(* CODESYS project Lauda.library
   Company: Ziga Javornik
   DefaultNamespace: ZigaLibs.Lauda
   Version: 0.0.2.2
   Placeholder: ZigaLibs.Lauda
   Author: Ziga Javornik
   Description: Various Lauda device implementations.
   Title: ZigaLibs.Lauda

Project tree, tasks and I/O mapping:
  libraries: Tc2_Standard, * (Beckhoff Automation GmbH); Tc2_System, * (Beckhoff Automation GmbH); Tc2_TcpIp, * (Beckhoff Automation GmbH); Tc2_Utilities, * (Beckhoff Automation GmbH); Tc3_Module, * (Beckhoff Automation GmbH); TcUnit, 1.3.1 (www.tcunit.org); ZigaLibs.Core, 0.0.3.7 (Ziga Javornik); TcpIp, 0.0.2.2 (Ziga Javornik); ZigaLibs.Logging, * (Ziga Javornik)
  GVLs/
  SOURCE/
    Lauda Pro P20/
      DUTs/
        Commands/
          Read/
            Command groups/
              data type ST_LaudaReadCommands_ActuatingSignal
              data type ST_LaudaReadCommands_Control
              data type ST_LaudaReadCommands_ControlParameters
              data type ST_LaudaReadCommands_Cooling
              data type ST_LaudaReadCommands_FillLevel
              data type ST_LaudaReadCommands_Pump
              data type ST_LaudaReadCommands_Rights
              data type ST_LaudaReadCommands_Safety
              data type ST_LaudaReadCommands_Status
              data type ST_LaudaReadCommands_SwVersions
              data type ST_LaudaReadCommands_Temperature
            data type ST_LaudaReadCommands
          Write/
            Command groups/
              data type ST_LaudaWriteCommands_Control
              data type ST_LaudaWriteCommands_ControlParameters
              data type ST_LaudaWriteCommands_Cooling
              data type ST_LaudaWriteCommands_Pump
              data type ST_LaudaWriteCommands_Rights
              data type ST_LaudaWriteCommands_Safety
              data type ST_LaudaWriteCommands_Status
              data type ST_LaudaWriteCommands_Temperature
            data type ST_LaudaWriteCommands
          data type ST_LaudaCommands
        Errors/
          data type E_LaudaResponseError
          data type ST_LaudaFaults
          data type ST_LaudaReadWriteError
          data type ST_LaudaResponseErrors
        Parameters/
          data type ST_LaudaActualValuesCollection
          data type ST_LaudaCommParameters
        States/
          data type E_LaudaParameterReadState
          data type E_LaudaParameterWriteState
          data type E_ReadWriteStep
      POUs/
        Helpers/
          function block FB_LaudaCommandGenerator [ST]: KeyboardMasterLock, KeyboardMasterUnlock, KeyboardRemoteUnitLock, KeyboardRemoteUnitUnlock, SafetyActivate, SafetyDeactivate, SetPumpStage, SetTemperature, Start, Stop
          program LaudaHelper [ST]: AddSuffix, GenerateComand, ParseLaudaFaultDiagnosis, ParseResponseError, RemoveSuffix, ValidateReadCommandResponse, ValidateSendCommandResponse, Commands, ResponseErrors
        function block FB_LaudaPro_P20 [ST]: FB_init, AddToErrorBuffer, DequeueCommand, EnqueueCommand, ActualValues, CommParameters, DeviceFaultDiagnosis, Error, ErrorBuffer, Faults, TcpIpConnectionEstablished
  TESTS/
    Test suites/
      function block FB_LaudaHelperTests [ST]: Test01_AddSuffix, Test02_RemoveSuffix, Test03_ValidateReadCommandResponse, Test04_ValidateSendCommandResponse, Test05_ParseFault, Test06_ParseResponseError
    program PRG_TESTS [ST]
*)

// SOURCE/Lauda Pro P20/DUTs/Commands/Read/Command groups/ST_LaudaReadCommands_ActuatingSignal
TYPE ST_LaudaReadCommands_ActuatingSignal :
STRUCT
	Value	: STRING := 'IN_PV_06';
END_STRUCT
END_TYPE

// SOURCE/Lauda Pro P20/DUTs/Commands/Read/Command groups/ST_LaudaReadCommands_Control
TYPE ST_LaudaReadCommands_Control :
STRUCT
	SetpointOffset	: STRING := 'IN_PAR_14_';
	ControlVariable	: STRING := 'IN_MODE_01';
	OffsetSource	: STRING := 'IN_MODE_04';
END_STRUCT
END_TYPE

// SOURCE/Lauda Pro P20/DUTs/Commands/Read/Command groups/ST_LaudaReadCommands_ControlParameters
TYPE ST_LaudaReadCommands_ControlParameters :
STRUCT
END_STRUCT
END_TYPE

// SOURCE/Lauda Pro P20/DUTs/Commands/Read/Command groups/ST_LaudaReadCommands_Cooling
TYPE ST_LaudaReadCommands_Cooling :
STRUCT
	CoolingMode	: STRING := 'IN_SP_02';
END_STRUCT
END_TYPE

// SOURCE/Lauda Pro P20/DUTs/Commands/Read/Command groups/ST_LaudaReadCommands_FillLevel
TYPE ST_LaudaReadCommands_FillLevel :
STRUCT
	BathLevel	: STRING := 'IN_PV_05';
END_STRUCT
END_TYPE

// SOURCE/Lauda Pro P20/DUTs/Commands/Read/Command groups/ST_LaudaReadCommands_Pump
TYPE ST_LaudaReadCommands_Pump :
STRUCT
	FlowRate	: STRING := 'IN_PV_07';
	PowerStage	: STRING := 'IN_SP_01';
END_STRUCT
END_TYPE

// SOURCE/Lauda Pro P20/DUTs/Commands/Read/Command groups/ST_LaudaReadCommands_Rights
TYPE ST_LaudaReadCommands_Rights :
STRUCT
	KeyboardMaster_Locked				: STRING := 'IN_MODE_00_';
	KeyboardRemoveControlUnit_Locked	: STRING := 'IN_MODE_03';
END_STRUCT
END_TYPE

// SOURCE/Lauda Pro P20/DUTs/Commands/Read/Command groups/ST_LaudaReadCommands_Safety
TYPE ST_LaudaReadCommands_Safety :
STRUCT
	CommTimeoutViaInterface : STRING := 'IN_SP_08';
	SafetyModeActive		: STRING := 'IN_MODE_06';
END_STRUCT
END_TYPE

// SOURCE/Lauda Pro P20/DUTs/Commands/Read/Command groups/ST_LaudaReadCommands_Status
TYPE ST_LaudaReadCommands_Status :
STRUCT
	StandBy			: STRING := 'IN_MODE_02';
	DeviceType		: STRING := 'TYPE';
	DeviceStatus	: STRING := 'STATUS';
	FaultDiagnosis	: STRING := 'STAT';
END_STRUCT
END_TYPE

// SOURCE/Lauda Pro P20/DUTs/Commands/Read/Command groups/ST_LaudaReadCommands_SwVersions
TYPE ST_LaudaReadCommands_SwVersions :
STRUCT
	ControlSyste							: STRING := 'VERSION_R';
	ProtectionSystem						: STRING := 'VERSION_S';
	RemoteControl							: STRING := 'VERSION_B';
	CoolingSystem							: STRING := 'VERSION_T';
	AnalogInterfaceModule					: STRING := 'VERSION_A';
	RS232_422_Profibus_Profinet				: STRING := 'VERSION_V';
	EtherCAT								: STRING := 'VERSION_Z';
	ContactInterace							: STRING := 'VERSION_D';
	SolenoidValveForCoolingWater			: STRING := 'VERSION_M_0';
	SolenoidValveForAutomaticFillingDevice	: STRING := 'VERSION_M_1';
	SolenoidValveForConstantLevelDevice		: STRING := 'VERSION_M_2';
	SolenoidValve_ShutOffValve1				: STRING := 'VERSION_M_3';
	SolenoidValve_ShutOffValve2				: STRING := 'VERSION_M_4';
	ExternalPT100_interface1				: STRING := 'VERSION_E';
END_STRUCT
END_TYPE

// SOURCE/Lauda Pro P20/DUTs/Commands/Read/Command groups/ST_LaudaReadCommands_Temperature
TYPE ST_LaudaReadCommands_Temperature :
STRUCT
	TemperatureSetpoint				: STRING	 := 'IN_SP_00';
	BathTemperatureOutflow_01C		: STRING	 := 'IN_PV_00';
	BathTemperatureOutflow_001C		: STRING	 := 'IN_PV_10';
	QueryControlledTemperature		: STRING	 := 'IN_PV_01';
	ExternalTemperature_Pt_C		: STRING	 := 'IN_PV_03';
	ExternalTemperature_AnalogInput	: STRING	 := 'IN_PV_04';
	ExternalTemperature_Pt_001_C	: STRING	 := 'IN_PV_13';
	OvertemperatureTurnoffPoint_Tmax: STRING	 := 'IN_SP_03';
	OutflowLimmitHigh				: STRING	 := 'IN_SP_04';
	OutflowLimmitLow				: STRING	 := 'IN_SP_05';
	SafetyModeTemperature 			: STRING	 := 'IN_SP_07';
END_STRUCT
END_TYPE

// SOURCE/Lauda Pro P20/DUTs/Commands/Read/ST_LaudaReadCommands
TYPE ST_LaudaReadCommands :
STRUCT
	Temperature			: ST_LaudaReadCommands_Temperature;
	Pump				: ST_LaudaReadCommands_Pump;
	FillLevel			: ST_LaudaReadCommands_FillLevel;
	ActuatingSignal		: ST_LaudaReadCommands_ActuatingSignal;
	Cooling				: ST_LaudaReadCommands_Cooling;
	Safety				: ST_LaudaReadCommands_Safety;
	ControlParameters	: ST_LaudaReadCommands_ControlParameters;
	Control				: ST_LaudaReadCommands_Control;
	Rights				: ST_LaudaReadCommands_Rights;
	Status				: ST_LaudaReadCommands_Status;
	SwVersion			: ST_LaudaReadCommands_SwVersions;	
END_STRUCT
END_TYPE

// SOURCE/Lauda Pro P20/DUTs/Commands/Write/Command groups/ST_LaudaWriteCommands_Control
TYPE ST_LaudaWriteCommands_Control :
STRUCT
	SetpointOffset	: STRING := 'OUT_PAR_14_';
	ControlVariable	: STRING := 'OUT_MODE_01_X';
	OffsetSource	: string := 'OUT_MODE_04_X';
END_STRUCT
END_TYPE

// SOURCE/Lauda Pro P20/DUTs/Commands/Write/Command groups/ST_LaudaWriteCommands_ControlParameters
TYPE ST_LaudaWriteCommands_ControlParameters :
STRUCT
	Xp						: STRING := 'OUT_PAR_00_';
	Tn						: STRING := 'OUT_PAR_01_';
	Tv						: STRING := 'OUT_PAR_02_';
	Td						: STRING := 'OUT_PAR_03_';
	KpE						: STRING := 'OUT_PAR_04_';
	TnE						: STRING := 'OUT_PAR_05_';
	TvE						: STRING := 'OUT_PAR_06_';
	TdE						: STRING := 'OUT_PAR_07_';
	CorrectionLimitation	: STRING := 'OUT_PAR_09_';
	XpF						: STRING := 'OUT_PAR_10_';
	Prop_E					: STRING := 'OUT_PAR_15_';
END_STRUCT
END_TYPE

// SOURCE/Lauda Pro P20/DUTs/Commands/Write/Command groups/ST_LaudaWriteCommands_Cooling
TYPE ST_LaudaWriteCommands_Cooling :
STRUCT
	CoolingMode	: STRING := 'OUT_SP_02';
END_STRUCT
END_TYPE

// SOURCE/Lauda Pro P20/DUTs/Commands/Write/Command groups/ST_LaudaWriteCommands_Pump
TYPE ST_LaudaWriteCommands_Pump :
STRUCT
	Stage	: STRING := 'OUT_SP_01_';	// Pump stage 1-6 or 1-8 (device specific)
END_STRUCT
END_TYPE

// SOURCE/Lauda Pro P20/DUTs/Commands/Write/Command groups/ST_LaudaWriteCommands_Rights
TYPE ST_LaudaWriteCommands_Rights :
STRUCT
	KeyboardMaster_UnlockLock				: STRING := 'OUT_MODE_00_';
	KeyboardRemoteControlUnit_UnlockLock	: STRING := 'OUT_MODE_03_';
END_STRUCT
END_TYPE

// SOURCE/Lauda Pro P20/DUTs/Commands/Write/Command groups/ST_LaudaWriteCommands_Safety
TYPE ST_LaudaWriteCommands_Safety :
STRUCT
	CommTimeoutViaInterface : STRING := 'OUT_SP_08_';
	ActivateSafetyMode		: STRING := 'OUT_MODE_06_';
END_STRUCT
END_TYPE

// SOURCE/Lauda Pro P20/DUTs/Commands/Write/Command groups/ST_LaudaWriteCommands_Status
TYPE ST_LaudaWriteCommands_Status :
STRUCT
	Start	: STRING := 'START';
	Stop	: STRING := 'STOP';
END_STRUCT
END_TYPE

// SOURCE/Lauda Pro P20/DUTs/Commands/Write/Command groups/ST_LaudaWriteCommands_Temperature
TYPE ST_LaudaWriteCommands_Temperature :
STRUCT
	TemperatureSet				: STRING := 'OUT_SP_00_';
	ActualExternalTemperature	: STRING := 'OUT_PV_05_';
	OutflowLimmitHigh			: STRING := 'OUT_SP_04_';
	OutflowLimmitLow			: STRING := 'OUT_SP_05_';
	SafetyModeTemperature		: STRING := 'OUT_SP_07_';
END_STRUCT
END_TYPE

// SOURCE/Lauda Pro P20/DUTs/Commands/Write/ST_LaudaWriteCommands
TYPE ST_LaudaWriteCommands :
STRUCT
	Temperature			: ST_LaudaWriteCommands_Temperature;
	Control				: ST_LaudaWriteCommands_Control;
	ControlParameters	: ST_LaudaWriteCommands_ControlParameters;
	Cooling				: ST_LaudaWriteCommands_Cooling;
	Pump				: ST_LaudaWriteCommands_Pump;
	Rights				: ST_LaudaWriteCommands_Rights;
	Safety				: ST_LaudaWriteCommands_Safety;
	Status				: ST_LaudaWriteCommands_Status;
END_STRUCT
END_TYPE

// SOURCE/Lauda Pro P20/DUTs/Commands/ST_LaudaCommands
TYPE ST_LaudaCommands :
STRUCT
	Read	: ST_LaudaReadCommands;
	Write	: ST_LaudaWriteCommands;
END_STRUCT
END_TYPE

// SOURCE/Lauda Pro P20/DUTs/Errors/E_LaudaResponseError
{attribute 'qualified_only'}
{attribute 'strict'}
TYPE E_LaudaResponseError :
(
	NO_ERROR := 0,
	WRONG_ENTRY,
	WRONG_COMMAND,
	SYNTAX_ERROR,
	IMPERMISSABLE_VALUE,
	MODULE_OR_VALUE_NOT_AVAILABLE,
	ALL_SEGMENTS_IN_THE_PROGRAMMER_OCCUPIED,
	SETPOINT_NOT_POSSIBLE_WITH_ANALOG_SETPOINT_USED,
	EXTERNAL_TEMPERATURE_PROBE_MISSING,
	ANALOG_VALUE_NOT_PRESENT,
	SAFETY_MODE_CANT_START_IF_NOT_ENABLED,
	CANT_SET_VALUE_PROGRAMMER_RUNNING_OR_PAUSED,
	CANT_START_PROGRAMMER_ANALOG_SETPOINT_USED,
	CANT_ACTIVATE_FROM_SAFETY_MODE);
END_TYPE

// SOURCE/Lauda Pro P20/DUTs/Errors/ST_LaudaFaults
{attribute 'qualified_only'}
{attribute 'strict'}
TYPE ST_LaudaFaults :
STRUCT
	Error						: BOOL;
	Alarm						: BOOL;
	Warning						: BOOL;
	Overtemp					: BOOL;
	Sublevel					: BOOL;
	HigherLevel					: BOOL;
	ExternalControlValueMissing	: BOOL;
END_STRUCT
END_TYPE

// SOURCE/Lauda Pro P20/DUTs/Errors/ST_LaudaReadWriteError
{attribute 'qualified_only'}
{attribute 'strict'}
TYPE ST_LaudaReadWriteError :
STRUCT
	SendCommand			: STRING(100);
	ResponseErrorInfo	: E_LaudaResponseError;
END_STRUCT
END_TYPE

// SOURCE/Lauda Pro P20/DUTs/Errors/ST_LaudaResponseErrors
{attribute 'qualified_only'}
{attribute 'strict'}
{attribute 'to_string'}
TYPE ST_LaudaResponseErrors :
STRUCT
	WrongEntry	 								: STRING := 'ERR_2';
	WrongCommand								: STRING := 'ERR_3';
	SyntaxError	 								: STRING := 'ERR_5';
	ImpermissableValue	 						: STRING := 'ERR_6';
	ModuleOrValueNotAvailable					: STRING := 'ERR_8';
	AllSegmentsInTheProgrammerAreOccupied		: STRING := 'ERR_30';
	SetpointNotPossible_AnalogSetpointIsUsed	: STRING := 'ERR_31';
	ExternalTemperatureProbeMissing	 			: STRING := 'ERR_33';
	AnalogValueNotPresent	 					: STRING := 'ERR_34';
	SafetyModeCantBeStarted_ItIsNotEnabled	 	: STRING := 'ERR_35';
	CantSetValue_ProgrammerRunningOrPaused	 	: STRING := 'ERR_36';
	CantStartProgrammer_AnalogSetpointIsUsed	: STRING := 'ERR_37';
	CantActivateFromSafetyMode	 				: STRING := 'ERR_38';
END_STRUCT
END_TYPE

// SOURCE/Lauda Pro P20/DUTs/Parameters/ST_LaudaActualValuesCollection
{attribute 'qualified_only'}
{attribute 'strict'}
TYPE ST_LaudaActualValuesCollection :
STRUCT
	BathTemperature		: REAL;
	TemperatureSetpoint	: REAL;
	PumpStage			: UINT;
	StandBy				: BOOL;
	LiquidLevel			: UINT;
END_STRUCT
END_TYPE

// SOURCE/Lauda Pro P20/DUTs/Parameters/ST_LaudaCommParameters
{attribute 'qualified_only'}
{attribute 'strict'}
TYPE ST_LaudaCommParameters :
STRUCT
	ReadCycle		: TIME := T#500MS;			// Cyclic reading of certain values is executed within the interval defined by this parameter.
	ReconnectPeriod	: TIME := T#45S;			// Reconnect period for TCP/IP. Don't set too low (30s should be the lowest)
	Ipv4Address		: Tc2_System.T_IPv4Addr;	// IPV4 address of the device.
	Port			: UINT;						// Port of the device.
END_STRUCT
END_TYPE

// SOURCE/Lauda Pro P20/DUTs/States/E_LaudaParameterReadState
{attribute 'qualified_only'}
{attribute 'strict'}
TYPE E_LaudaParameterReadState :
(
	READY := 0,
	ACTUAL_TEMPERATURE_SETPOINT,
	BAH_OUTFLOW_TEMP,
	PUMP_STAGE,
	READ_ENABLE_STATE,
	OIL_LEVEL,
	FAULT_DIAGNOSIS,
	DONE
);
END_TYPE

// SOURCE/Lauda Pro P20/DUTs/States/E_LaudaParameterWriteState
{attribute 'qualified_only'}
{attribute 'strict'}
TYPE E_LaudaParameterWriteState :
(
	READY,
	SEND,
	AWAIT_RESPONSE,
	VALIDATE_RESPONSE,
	DONE
);
END_TYPE

// SOURCE/Lauda Pro P20/DUTs/States/E_ReadWriteStep
{attribute 'qualified_only'}
{attribute 'strict'}
TYPE E_ReadWriteStep :
(
	SEND,
	AWAIT_RESPONSE
);
END_TYPE

// SOURCE/Lauda Pro P20/POUs/Helpers/FB_LaudaCommandGenerator
FUNCTION_BLOCK FB_LaudaCommandGenerator
VAR_INPUT
END_VAR
VAR_OUTPUT
END_VAR
VAR
	_formatString	: Tc2_Utilities.FB_FormatString;
END_VAR

METHOD KeyboardMasterLock : T_MaxString
VAR_INPUT
END_VAR
KeyboardMasterLock := LaudaHelper.AddSuffix(CONCAT(
	STR1 := LaudaHelper.Commands.Write.Rights.KeyboardMaster_UnlockLock, 
	STR2 := '1'));
END_METHOD

METHOD KeyboardMasterUnlock : T_MaxString
VAR_INPUT
END_VAR
KeyboardMasterUnlock := LaudaHelper.AddSuffix(CONCAT(
	STR1 := LaudaHelper.Commands.Write.Rights.KeyboardMaster_UnlockLock, 
	STR2 := '0'));
END_METHOD

METHOD KeyboardRemoteUnitLock : Tc2_System.T_MaxString
VAR_INPUT
END_VAR
KeyboardRemoteUnitLock := LaudaHelper.AddSuffix(CONCAT(
	STR1 := LaudaHelper.Commands.Write.Rights.KeyboardRemoteControlUnit_UnlockLock, 
	STR2 := '1'));
END_METHOD

METHOD KeyboardRemoteUnitUnlock : Tc2_System.T_MaxString
VAR_INPUT
END_VAR
KeyboardRemoteUnitUnlock := LaudaHelper.AddSuffix(CONCAT(
	STR1 := LaudaHelper.Commands.Write.Rights.KeyboardRemoteControlUnit_UnlockLock, 
	STR2 := '0'));
END_METHOD

// Activates safety mode.
METHOD PUBLIC SafetyActivate : T_MaxString
VAR_INPUT
END_VAR
SafetyActivate := LaudaHelper.AddSuffix(
	sData := CONCAT(STR1 := LaudaHelper.Commands.Write.Safety.ActivateSafetyMode, STR2 := '1'));
END_METHOD

// Deactivates safety mode
METHOD PUBLIC SafetyDeactivate : T_MaxString
VAR_INPUT
END_VAR
SafetyDeactivate := LaudaHelper.AddSuffix(
	sData := CONCAT(STR1 := LaudaHelper.Commands.Write.Safety.ActivateSafetyMode, STR2 := '0'));
END_METHOD

// Sets pump stage, 1-6/9, depending on device specification
METHOD PUBLIC SetPumpStage : T_MaxString
VAR_INPUT
	nStage	: UINT;
END_VAR

VAR
	nPumpStageWithLimits	: UINT;
END_VAR
IF nStage < 1 THEN
	nPumpStageWithLimits := 1;
ELSIF nStage > 8 THEN
	nPumpStageWithLimits := 8;
ELSE
	nPumpStageWithLimits := nStage;
END_IF

SetPumpStage := LaudaHelper.AddSuffix(sData := Tc2_Standard.CONCAT(
		STR1 := LaudaHelper.Commands.Write.Pump.Stage, 
		STR2 := UINT_TO_STRING(nPumpStageWithLimits)));
END_METHOD

// Creates the command for temperature setting.
METHOD PUBLIC SetTemperature : T_maxstring
VAR_INPUT
	fTemperature	: REAL;	// Temperature setpoint to be set on the device.
END_VAR

VAR_INST
	errorID	: UDINT;
END_VAR
_formatString(
	sFormat := CONCAT(LaudaHelper.Commands.Write.Temperature.TemperatureSet, '%06.2f'),
	arg1 := Tc2_Utilities.F_REAL(in := fTemperature),
	nErrId => errorID);

SetTemperature := LaudaHelper.AddSuffix(_formatString.sOut);
END_METHOD

// Starts the device
METHOD PUBLIC Start : T_MaxString
Start := LaudaHelper.AddSuffix(sData := LaudaHelper.Commands.Write.Status.Start);
END_METHOD

// Stops the device
METHOD PUBLIC Stop : T_MaxString
Stop := LaudaHelper.AddSuffix(sData := LaudaHelper.Commands.Write.Status.Stop);
END_METHOD

END_FUNCTION_BLOCK

// SOURCE/Lauda Pro P20/POUs/Helpers/LaudaHelper
{attribute 'no_explicit_call' := 'Body contains no logic, calling methods only allowed.'}
{attribute 'hide_all_locals'}
// Provides various helper methods for easier communication with Lauda Pro device. 
// Program does not require being called, a simple access to methods is enough.
PROGRAM LaudaHelper
VAR
	_formatString			: FB_FormatString;
	_laudaCommandGenerator	: FB_LaudaCommandGenerator;	
	_commands				: ST_LaudaCommands;
	_responseErrors			: ST_LaudaResponseErrors;
END_VAR

VAR CONSTANT
	COMMAND_SUFFIX				: STRING := '$R$L';
	SEND_COMMAND_RESPONSE_OK	: STRING := 'OK';
	COMMAND_RESPONSE_ERROR		: STRING := 'ERR_'; 
END_VAR

// Adds suffix to the data command.
METHOD PUBLIC AddSuffix : Tc2_System.T_MaxString
VAR_INPUT
	sData	: Tc2_System.T_MaxString;
END_VAR
AddSuffix := Tc2_Standard.CONCAT(STR1 := sData, STR2 := COMMAND_SUFFIX);
END_METHOD

// Provides access to command generation methods.
METHOD PUBLIC GenerateComand : REFERENCE TO FB_LaudaCommandGenerator
VAR_INPUT
END_VAR
GenerateComand ref= _laudaCommandGenerator;
END_METHOD

// Parses the RAW data response for fault diagnosis and returns the faults structure.
METHOD ParseLaudaFaultDiagnosis : ST_LaudaFaults
VAR_INPUT
	sDiagnosisResposne	: Tc2_System.T_MaxString;
END_VAR
VAR
	sTmp		: Tc2_System.T_MaxString;
	nResponse	: BYTE;
	stFaults	: ST_LaudaFaults;
END_VAR

(*

*)
sTmp := RemoveSuffix(sData := sDiagnosisResposne);

stFaults.Error := INT_TO_BOOL(STRING_TO_INT(Tc2_Standard.MID(
	STR := sTmp,
	POS := 1, 
	LEN := 1)));

stFaults.Alarm := INT_TO_BOOL(STRING_TO_INT(Tc2_Standard.MID(
	STR := sTmp,
	POS := 2, 
	LEN := 1)));
	
stFaults.Warning := INT_TO_BOOL(STRING_TO_INT(Tc2_Standard.MID(
	STR := sTmp,
	POS := 3, 
	LEN := 1)));
	
stFaults.Overtemp := INT_TO_BOOL(STRING_TO_INT(Tc2_Standard.MID(
	STR := sTmp,
	POS := 4, 
	LEN := 1)));
	
stFaults.Sublevel := INT_TO_BOOL(STRING_TO_INT(Tc2_Standard.MID(
	STR := sTmp,
	POS := 5, 
	LEN := 1)));
	
stFaults.HigherLevel := INT_TO_BOOL(STRING_TO_INT(Tc2_Standard.MID(
	STR := sTmp,
	POS := 6, 
	LEN := 1)));
	
stFaults.ExternalControlValueMissing := INT_TO_BOOL(STRING_TO_INT(Tc2_Standard.MID(
	STR := sTmp,
	POS := 7, 
	LEN := 1)));
	
ParseLaudaFaultDiagnosis := stFaults;
END_METHOD

// Parses the error and returns the error message for further diagnosis
METHOD PUBLIC ParseResponseError : E_LaudaResponseError
VAR_INPUT
	Response	: Tc2_System.T_MaxString;
END_VAR
// Search the errors from highest to lowest to avoid case such as ERR_30 and you find it with ERR_3
// If success, return
IF Tc2_Standard.FIND(
	STR1 := Response, 
	STR2 := ResponseErrors.CantActivateFromSafetyMode) <> 0 
THEN
	ParseResponseError := E_LaudaResponseError.CANT_ACTIVATE_FROM_SAFETY_MODE;
	RETURN;
END_IF

IF Tc2_Standard.FIND(
	STR1 := Response, 
	STR2 := ResponseErrors.CantStartProgrammer_AnalogSetpointIsUsed) <> 0 
THEN
	ParseResponseError :=  E_LaudaResponseError.CANT_START_PROGRAMMER_ANALOG_SETPOINT_USED;
	RETURN;
END_IF

IF Tc2_Standard.FIND(
	STR1 := Response, 
	STR2 := ResponseErrors.CantSetValue_ProgrammerRunningOrPaused) <> 0 
THEN
	ParseResponseError :=  E_LaudaResponseError.CANT_SET_VALUE_PROGRAMMER_RUNNING_OR_PAUSED;
	RETURN;
END_IF

IF Tc2_Standard.FIND(
	STR1 := Response, 
	STR2 := ResponseErrors.SafetyModeCantBeStarted_ItIsNotEnabled) <> 0 
THEN
	ParseResponseError := E_LaudaResponseError.SAFETY_MODE_CANT_START_IF_NOT_ENABLED;
	RETURN;
END_IF

IF Tc2_Standard.FIND(
	STR1 := Response, 
	STR2 := ResponseErrors.AnalogValueNotPresent) <> 0 
THEN
	ParseResponseError := E_LaudaResponseError.ANALOG_VALUE_NOT_PRESENT;
	RETURN;
END_IF

IF Tc2_Standard.FIND(
	STR1 := Response, 
	STR2 := ResponseErrors.ExternalTemperatureProbeMissing) <> 0 
THEN
	ParseResponseError := E_LaudaResponseError.EXTERNAL_TEMPERATURE_PROBE_MISSING;
	RETURN;
END_IF

IF Tc2_Standard.FIND(
	STR1 := Response, 
	STR2 := ResponseErrors.SetpointNotPossible_AnalogSetpointIsUsed) <> 0 
THEN
	ParseResponseError := E_LaudaResponseError.SETPOINT_NOT_POSSIBLE_WITH_ANALOG_SETPOINT_USED;
	RETURN;
END_IF

IF Tc2_Standard.FIND(
	STR1 := Response, 
	STR2 := ResponseErrors.AllSegmentsInTheProgrammerAreOccupied) <> 0 
THEN
	ParseResponseError := E_LaudaResponseError.ALL_SEGMENTS_IN_THE_PROGRAMMER_OCCUPIED;
	RETURN;
END_IF

IF Tc2_Standard.FIND(
	STR1 := Response, 
	STR2 := ResponseErrors.ModuleOrValueNotAvailable) <> 0 
THEN
	ParseResponseError := E_LaudaResponseError.MODULE_OR_VALUE_NOT_AVAILABLE;
	RETURN;
END_IF

IF Tc2_Standard.FIND(
	STR1 := Response, 
	STR2 := ResponseErrors.ImpermissableValue) <> 0 
THEN
	ParseResponseError := E_LaudaResponseError.IMPERMISSABLE_VALUE;
	RETURN;
END_IF

IF Tc2_Standard.FIND(
	STR1 := Response, 
	STR2 := ResponseErrors.SyntaxError) <> 0 
THEN
	ParseResponseError := E_LaudaResponseError.SYNTAX_ERROR;
	RETURN;
END_IF

IF Tc2_Standard.FIND(
	STR1 := Response, 
	STR2 := ResponseErrors.WrongCommand) <> 0 
THEN
	ParseResponseError := E_LaudaResponseError.WRONG_COMMAND;
	RETURN;
END_IF

IF Tc2_Standard.FIND(
	STR1 := Response, 
	STR2 := ResponseErrors.WrongEntry) <> 0 
THEN
	ParseResponseError := E_LaudaResponseError.WRONG_ENTRY;
	RETURN;
END_IF
END_METHOD

// Removes suffix from the provided data string
METHOD PUBLIC RemoveSuffix : Tc2_System.T_MaxString
VAR_INPUT
	sData	: Tc2_System.T_MaxString;
END_VAR

VAR
	sDataWithoutSuffix	: Tc2_System.T_MaxString;
END_VAR
Tc2_Utilities.FindAndDelete(
	pDstString := ADR(sDataWithoutSuffix),
	nDstSize := SIZEOF(sDataWithoutSuffix),
	pDeleteString := ADR(COMMAND_SUFFIX),
	pSrcString := ADR(sData));
	
RemoveSuffix := sDataWithoutSuffix;
END_METHOD

// Validates the response when doing a read command to Lauda Pro Thermostat.
// Returns TRUE if response is valid, or FALSE if it is not valid or an error was reported.
METHOD PUBLIC ValidateReadCommandResponse : BOOL
VAR_INPUT
	sResponse	: Tc2_System.T_MaxString;
END_VAR
ValidateReadCommandResponse := 
	Tc2_Standard.FIND(STR1 := sResponse, STR2 := COMMAND_RESPONSE_ERROR) = 0 AND
	Tc2_Standard.FIND(STR1 := sResponse, STR2 := COMMAND_SUFFIX) <> 0;
END_METHOD

// Validates the response when doing a write command to Lauda Pro Thermostat.
// Returns TRUE if response is valid, or FALSE if it is not valid or an error was reported
METHOD PUBLIC ValidateSendCommandResponse : BOOL
VAR_INPUT
	sResponse	: Tc2_System.T_MaxString;
END_VAR
ValidateSendCommandResponse := 
	Tc2_Standard.FIND(STR1 := sResponse, STR2 := SEND_COMMAND_RESPONSE_OK) <> 0 AND
	Tc2_Standard.FIND(STR1 := sResponse, STR2 := COMMAND_RESPONSE_ERROR) = 0 AND
	Tc2_Standard.FIND(STR1 := sResponse, STR2 := COMMAND_SUFFIX) <> 0;
END_METHOD

PROPERTY Commands : REFERENCE TO ST_LaudaCommands
GET
Commands ref= _commands;
END_GET
END_PROPERTY

PROPERTY ResponseErrors : REFERENCE TO ST_LaudaResponseErrors
GET
ResponseErrors ref= _responseErrors;
END_GET
END_PROPERTY

END_PROGRAM

// SOURCE/Lauda Pro P20/POUs/FB_LaudaPro_P20
(* LaudaPro P20 control via TCP/IP
Includes constructor parameters:
 - nMaxPumpLevel	: UINT;	// Max pump setting, value ranges from 1-6/8 depending on the device type*)
 
FUNCTION_BLOCK FB_LaudaPro_P20 EXTENDS ZigaLibs_Core.FB_HasInstanceNameAndPath

VAR_INPUT
	fTemperatureSet	: REAL;	// Temperature setpoint
	bSafetyOk		: BOOL;	// Safety mode actiation when FALSE
	bEnable			: BOOL;	// Enable temperature setting
	nPumpStage		: UINT := 2;	// Set pump stage 1-8
	bConnect		: BOOL;	// Connects to the device via TCP or disconnects if set to FALSE
	bKeyboardUnlock	: BOOL;	// Unlocks keyboard control
	bResendValues	: BOOL;	// Resends all current values to the device
	logger			: REFERENCE TO ZigaLibs_Logging.I_Logger;
END_VAR

VAR
	fbTcpIpControl		: ZigaLibs_TcpIp.FB_TcpIpCommControl(logger);
	TonReconnectTimer	: Tc2_Standard.TON;
	bFirstExecution		: BOOL := TRUE;

	// Writing
	fPrevTemperatureSet		: REAL;
	bPrevSafetyOk			: BOOL;
	bPrevEnable				: BOOL;
	nPrevPumpStage			: UINT;
	bPrevKeyboardUnlock		: BOOL;
	RtrigResendValues		: Tc2_Standard.R_TRIG;
	eWriteParameterState	: E_LaudaParameterWriteState;
	sWriteResponse			: Tc2_System.T_MaxString;
	arrCommandBuffer		: ARRAY[0..100] OF Tc2_System.T_MaxString;
	
	// Reading
	TonReadCycleTimer		: Tc2_Standard.TON;
	eReadParametersState	: E_LaudaParameterReadState;
	eReadParametersSubStep	: E_ReadWriteStep;
	sReadResponseString		: Tc2_System.T_MaxString;
	arrReadBufferErrors		: ARRAY[0..100] OF ST_LaudaReadWriteError;
	sCurrentReadCommand		: STRING;
	TonDelayReading			: Tc2_Standard.TON := (PT := T#100MS);
	TonDelayAwaitResponse	: Tc2_Standard.TON := (PT := T#100MS);
	// Logging
	bLoggerProvided			: BOOL;
	fbStringBuilder			: ZigaLibs_Core.FB_StringBuilder;
	
	// Property access fields
	_actualValues				: ST_LaudaActualValuesCollection;	// Actual values, reported back from the unit
	_error						: BOOL;	// Error flag
	_tcpIpConnectionEstablished	: BOOL;	// Connection indicator
	_commParameters				: ST_LaudaCommParameters;	// Parameters for TcpIp connection
	_maxPumpLevel				: UINT;
	_faults						: ST_LaudaFaults;
	_errorBuffer				: ARRAY[0..100] OF ST_LaudaReadWriteError;
END_VAR

VAR CONSTANT
	ABSOLUTE_MAX_PUMP_LEVEL : UINT := 8;	// The highest possible setting for pump is 8 for any device of this series
END_VAR

_error := FALSE;
bLoggerProvided := __ISVALIDREF(logger);

TonReconnectTimer(IN := NOT TonReconnectTimer.Q, PT := _commParameters.ReconnectPeriod);
RtrigResendValues(CLK := bResendValues);

// Set reconnect period
fbTcpIpControl.ReconnectPeriod := _commParameters.ReconnectPeriod;
fbTcpIpControl();

IF bConnect THEN
	// Connect/disconnect/error	
	IF fbTcpIpControl.Error AND TonReconnectTimer.Q THEN
		fbTcpIpControl.Disconnect();
	ELSIF fbTcpIpControl.IsConnected = FALSE THEN
		fbTcpIpControl.Connect(Ipv4Address := _commParameters.Ipv4Address, Port := _commParameters.Port);
	END_IF
ELSE
	fbTcpIpControl.Disconnect();
END_IF


IF fbTcpIpControl.Error THEN
	_error := TRUE;
END_IF

_tcpIpConnectionEstablished := fbTcpIpControl.IsConnected;
IF NOT _tcpIpConnectionEstablished THEN
	RETURN;
END_IF

//============================================================================
//======================= WRITE VALUES ON REQUEST ============================
//============================================================================

// Temperature setpoint
IF fPrevTemperatureSet <> fTemperatureSet OR bFirstExecution OR RtrigResendValues.Q THEN
	IF bLoggerProvided THEN
		fbStringBuilder.Reset()
			.AddString(str := THIS^.InstanceName)
			.AddString(str := ': Temperature setpoint changed from ')
			.AddWithDblQuotationMarks(str := REAL_TO_STRING(fPrevTemperatureSet))
			.AddString(str := ' to ')
 			.AddWithDblQuotationMarks(str := REAL_TO_STRING(fTemperatureSet))
			.AddString('.');
		logger.LogInfo(message := fbStringBuilder.Create());
	END_IF
	EnqueueCommand(Command :=
		LaudaHelper.GenerateComand().SetTemperature(fTemperature := fTemperatureSet));
END_IF

// Enable/Disable
IF bPrevEnable <> bEnable OR bFirstExecution OR RtrigResendValues.Q THEN
	IF bEnable THEN
		IF bLoggerProvided THEN
			fbStringBuilder.Reset()
				.AddString(str := THIS^.InstanceName)
				.AddString(str := ': Starting heating and pump operation.');
			logger.LogInfo(message := fbStringBuilder.Create());
		END_IF
		EnqueueCommand(Command := LaudaHelper.AddSuffix(LaudaHelper.Commands.Write.Status.Start));
	ELSE
		IF bLoggerProvided THEN
			fbStringBuilder.Reset()
				.AddString(str := THIS^.InstanceName)
				.AddString(str := ': Device is now stopped. Heating is stopped and pump is disabled.');
			logger.LogInfo(message := fbStringBuilder.Create());
		END_IF
		EnqueueCommand(Command := LaudaHelper.AddSuffix(LaudaHelper.Commands.Write.Status.Stop));	
	END_IF	
END_IF

// Safety
IF bPrevSafetyOk <> bSafetyOk OR bFirstExecution OR RtrigResendValues.Q THEN
	IF bSafetyOk THEN
		EnqueueCommand(LaudaHelper.GenerateComand().SafetyDeactivate());
	ELSE
		EnqueueCommand(LaudaHelper.GenerateComand().SafetyActivate());
	END_IF
END_IF

// Pump stage, limited between 1 and max value (6/8)
IF nPrevPumpStage <> nPumpStage OR bFirstExecution OR RtrigResendValues.Q THEN
	IF bLoggerProvided THEN
		fbStringBuilder.Reset()
			.AddString(str := THIS^.InstanceName)
			.AddString(str := ': Pump stage setting changed from ')
			.AddWithDblQuotationMarks(str := UINT_TO_STRING(nPrevPumpStage))
			.AddString(str := ' to ')
 			.AddWithDblQuotationMarks(str := UINT_TO_STRING(nPumpStage))
			.AddString('.');
		logger.LogInfo(message := fbStringBuilder.Create());
	END_IF
	EnqueueCommand(LaudaHelper.GenerateComand()
		.SetPumpStage(nStage := MIN(MAX(nPumpStage, 1), _maxPumpLevel)));
END_IF

// Keyobard locking
IF bPrevKeyboardUnlock <> bKeyboardUnlock OR bFirstExecution OR RtrigResendValues.Q THEN
	IF bKeyboardUnlock THEN
		EnqueueCommand(Command := LaudaHelper.GenerateComand().KeyboardMasterUnlock());
		EnqueueCommand(Command := LaudaHelper.GenerateComand().KeyboardRemoteUnitUnlock());
		IF bLoggerProvided THEN
			fbStringBuilder.Reset()
				.AddString(str := THIS^.InstanceName)
				.AddString(str := ': Keyboard changed from locked to unlocked.');
			logger.LogInfo(message := fbStringBuilder.Create());
		END_IF
	ELSE
		EnqueueCommand(Command := LaudaHelper.GenerateComand().KeyboardMasterLock());
		EnqueueCommand(Command := LaudaHelper.GenerateComand().KeyboardRemoteUnitLock());
		IF bLoggerProvided THEN
			fbStringBuilder.Reset()
				.AddString(str := THIS^.InstanceName)
				.AddString(str := ': Keyboard changed from unlocked to locked.');
			logger.LogInfo(message := fbStringBuilder.Create());
		END_IF
	END_IF
END_IF

bFirstExecution := FALSE;

// Only allow TCP/IP send/receive if connection is established. Exit the FB if connection is not valid to allow for a reset of TcpIp to go trough.
IF NOT _tcpIpConnectionEstablished THEN
	RETURN;
END_IF

// Write parameters from buffer
CASE eWriteParameterState OF
	E_LaudaParameterWriteState.READY:
		IF arrCommandBuffer[0] <> '' AND eReadParametersState = E_LaudaParameterReadState.READY THEN
			eWriteParameterState := E_LaudaParameterWriteState.SEND;
		END_IF
	
	E_LaudaParameterWriteState.SEND:
		IF NOT fbTcpIpControl.Error AND fbTcpIpControl.Send(arrCommandBuffer[0]) THEN
			eWriteParameterState := E_LaudaParameterWriteState.AWAIT_RESPONSE;
		END_IF
		
	 E_LaudaParameterWriteState.AWAIT_RESPONSE:
		 IF fbTcpIpControl.Receive(refResponse := sWriteResponse) THEN
			 eWriteParameterState := E_LaudaParameterWriteState.VALIDATE_RESPONSE;
		 END_IF
	 
	E_LaudaParameterWriteState.VALIDATE_RESPONSE:
		IF NOT LaudaHelper.ValidateSendCommandResponse(sResponse := sWriteResponse) THEN
			AddToErrorBuffer(sendCommand := arrCommandBuffer[0], response := sWriteResponse);
		END_IF

		DequeueCommand();
		eWriteParameterState := E_LaudaParameterWriteState.READY;
END_CASE

fPrevTemperatureSet := fTemperatureSet;
bPrevEnable := bEnable;
bPrevSafetyOk := bSafetyOk;
nPrevPumpStage := nPumpStage;
bPrevKeyboardUnlock := bKeyboardUnlock;

//============================================================================
//======================= READ VALUES CYCLICALLY =============================
//============================================================================

// Delay command send to wait for device to send correct data, some issues when sending commands too fast
TonDelayReading(
	IN := eReadParametersSubStep = E_ReadWriteStep.SEND);
TonDelayAwaitResponse(
	IN := eReadParametersSubStep = E_ReadWriteStep.AWAIT_RESPONSE);
TonReadCycleTimer(
	IN := TRUE, 
	PT := _commParameters.ReadCycle);

CASE eReadParametersState OF
	E_LaudaParameterReadState.READY:
		TonReadCycleTimer.IN := TRUE;
		IF eWriteParameterState = E_LaudaParameterWriteState.READY AND TonReadCycleTimer.Q THEN
			TonReadCycleTimer(IN := FALSE, PT := _commParameters.ReadCycle);
			eReadParametersSubStep := E_ReadWriteStep.SEND;
			eReadParametersState := E_LaudaParameterReadState.BAH_OUTFLOW_TEMP;
		END_IF
		
	E_LaudaParameterReadState.BAH_OUTFLOW_TEMP:
		CASE eReadParametersSubStep OF
			E_ReadWriteStep.SEND:
				IF TonDelayReading.Q THEN
					sCurrentReadCommand := LaudaHelper.AddSuffix(LaudaHelper.Commands.Read.Temperature.BathTemperatureOutflow_01C);
					IF fbTcpIpControl.Send(sCurrentReadCommand) THEN
						eReadParametersSubStep := E_ReadWriteStep.AWAIT_RESPONSE;			
					END_IF
				END_IF
				
			E_ReadWriteStep.AWAIT_RESPONSE:
				IF TonDelayAwaitResponse.Q THEN
					IF fbTcpIpControl.Receive(refResponse := sReadResponseString) THEN
						IF LaudaHelper.ValidateReadCommandResponse(sResponse := sReadResponseString) THEN
							_actualValues.BathTemperature := STRING_TO_REAL(LaudaHelper.RemoveSuffix(sReadResponseString));
						ELSE
							AddToErrorBuffer(response := sReadResponseString, sendCommand := sCurrentReadCommand);
						END_IF
						eReadParametersSubStep := E_ReadWriteStep.SEND;
						eReadParametersState := E_LaudaParameterReadState.ACTUAL_TEMPERATURE_SETPOINT;
					END_IF
				END_IF
		END_CASE

	E_LaudaParameterReadState.ACTUAL_TEMPERATURE_SETPOINT:
		CASE eReadParametersSubStep OF
			E_ReadWriteStep.SEND:
				IF TonDelayReading.Q THEN
					sCurrentReadCommand := LaudaHelper.AddSuffix(LaudaHelper.Commands.Read.Temperature.TemperatureSetpoint);
					IF fbTcpIpControl.Send(sCurrentReadCommand) THEN
						eReadParametersSubStep := E_ReadWriteStep.AWAIT_RESPONSE;			
					END_IF
				END_IF
				
			E_ReadWriteStep.AWAIT_RESPONSE:
				IF TonDelayAwaitResponse.Q THEN
					IF fbTcpIpControl.Receive(refResponse := sReadResponseString) THEN
						IF LaudaHelper.ValidateReadCommandResponse(sResponse := sReadResponseString) THEN
							_actualValues.TemperatureSetpoint := STRING_TO_REAL(LaudaHelper.RemoveSuffix(sReadResponseString));
						ELSE
							AddToErrorBuffer(response := sReadResponseString, sendCommand := sCurrentReadCommand);
						END_IF
						eReadParametersSubStep := E_ReadWriteStep.SEND;
						eReadParametersState := E_LaudaParameterReadState.PUMP_STAGE;
					END_IF
				END_IF
		END_CASE

		
	E_LaudaParameterReadState.PUMP_STAGE:
		CASE eReadParametersSubStep OF
			E_ReadWriteStep.SEND:
				IF TonDelayReading.Q THEN
					sCurrentReadCommand := LaudaHelper.AddSuffix(LaudaHelper.Commands.Read.Pump.PowerStage);
					IF fbTcpIpControl.Send(sCommand := sCurrentReadCommand) THEN
						eReadParametersSubStep := E_ReadWriteStep.AWAIT_RESPONSE;			
					END_IF
				END_IF
				
			E_ReadWriteStep.AWAIT_RESPONSE:
				IF TonDelayAwaitResponse.Q THEN
					IF fbTcpIpControl.Receive(refResponse := sReadResponseString) THEN
						IF LaudaHelper.ValidateReadCommandResponse(sResponse := sReadResponseString) THEN
							_actualValues.PumpStage := STRING_TO_UINT(Tc2_Standard.LEFT(
								STR := LaudaHelper.RemoveSuffix(sReadResponseString), 
								SIZE := 1));
						ELSE
							AddToErrorBuffer(response := sReadResponseString, sendCommand := sCurrentReadCommand);
						END_IF
						eReadParametersState := E_LaudaParameterReadState.READ_ENABLE_STATE;
						eReadParametersSubStep := E_ReadWriteStep.SEND;
					END_IF
				END_IF
		END_CASE
	
	E_LaudaParameterReadState.READ_ENABLE_STATE:
		CASE eReadParametersSubStep OF
			E_ReadWriteStep.SEND:
				IF TonDelayReading.Q THEN
					sCurrentReadCommand := LaudaHelper.AddSuffix(LaudaHelper.Commands.Read.Status.StandBy);
					IF fbTcpIpControl.Send(sCurrentReadCommand) THEN
						eReadParametersSubStep := E_ReadWriteStep.AWAIT_RESPONSE;			
					END_IF
				END_IF
				
			E_ReadWriteStep.AWAIT_RESPONSE:
				IF TonDelayAwaitResponse.Q THEN
					IF fbTcpIpControl.Receive(refResponse := sReadResponseString) THEN
						IF LaudaHelper.ValidateReadCommandResponse(sResponse := sReadResponseString) THEN
							_actualValues.StandBy := STRING_TO_BOOL(LaudaHelper.RemoveSuffix(sReadResponseString));
						ELSE
							AddToErrorBuffer(response := sReadResponseString, sendCommand := sCurrentReadCommand);
						END_IF
						eReadParametersSubStep := E_ReadWriteStep.SEND;
						eReadParametersState := E_LaudaParameterReadState.OIL_LEVEL;
					END_IF
				END_IF
		END_CASE
	
	E_LaudaParameterReadState.OIL_LEVEL:
		CASE eReadParametersSubStep OF
			E_ReadWriteStep.SEND:
				IF TonDelayReading.Q THEN
					sCurrentReadCommand :=  LaudaHelper.AddSuffix(LaudaHelper.Commands.Read.FillLevel.BathLevel);
					IF fbTcpIpControl.Send(sCommand := sCurrentReadCommand) THEN
						eReadParametersSubStep := E_ReadWriteStep.AWAIT_RESPONSE;			
					END_IF
				END_IF
				
			E_ReadWriteStep.AWAIT_RESPONSE:
				IF TonDelayAwaitResponse.Q THEN
					IF fbTcpIpControl.Receive(refResponse := sReadResponseString) THEN
						IF LaudaHelper.ValidateReadCommandResponse(sResponse := sReadResponseString) THEN
							_actualValues.LiquidLevel := STRING_TO_UINT(LaudaHelper.RemoveSuffix(sReadResponseString));
						ELSE
							AddToErrorBuffer(response := sReadResponseString, sendCommand := sCurrentReadCommand);
						END_IF
						eReadParametersState := E_LaudaParameterReadState.FAULT_DIAGNOSIS;
						eReadParametersSubStep := E_ReadWriteStep.SEND;
					END_IF
				END_IF
		END_CASE
		
	E_LaudaParameterReadState.FAULT_DIAGNOSIS:
		CASE eReadParametersSubStep OF
			E_ReadWriteStep.SEND:
				IF TonDelayReading.Q THEN
					sCurrentReadCommand := LaudaHelper.AddSuffix(LaudaHelper.Commands.Read.Status.FaultDiagnosis);
					IF fbTcpIpControl.Send(sCurrentReadCommand) THEN
						eReadParametersSubStep := E_ReadWriteStep.AWAIT_RESPONSE;			
					END_IF
				END_IF
				
			E_ReadWriteStep.AWAIT_RESPONSE:
				IF TonDelayAwaitResponse.Q THEN
					IF fbTcpIpControl.Receive(refResponse := sReadResponseString) THEN
						IF LaudaHelper.ValidateReadCommandResponse(sResponse := sReadResponseString) THEN
							_faults := LaudaHelper.ParseLaudaFaultDiagnosis(sDiagnosisResposne := sReadResponseString);
						ELSE
							AddToErrorBuffer(response := sReadResponseString, sendCommand := sCurrentReadCommand);
						END_IF
						eReadParametersState := E_LaudaParameterReadState.DONE;
						eReadParametersSubStep := E_ReadWriteStep.SEND;
					END_IF
				END_IF
		END_CASE	
		
	E_LaudaParameterReadState.DONE:
		eReadParametersState := E_LaudaParameterReadState.READY;
END_CASE

METHOD FB_init : BOOL
VAR_INPUT
	bInitRetains : BOOL; // if TRUE, the retain variables are initialized (warm start / cold start)
	bInCopyCode : BOOL;  // if TRUE, the instance afterwards gets moved into the copy code (online change)
	nMaxPumpLevel	: UINT;	// Max pump setting, value ranges from 1-6/8 depending on the device type
END_VAR
IF nMaxPumpLevel <= ABSOLUTE_MAX_PUMP_LEVEL THEN
	_maxPumpLevel := nMaxPumpLevel;
ELSE
	_maxPumpLevel := ABSOLUTE_MAX_PUMP_LEVEL;
END_IF
END_METHOD

// Adds the data to the error buffer and sets the _error to TRUE
METHOD PRIVATE AddToErrorBuffer
VAR_INPUT
	sendCommand	: Tc2_System.T_MaxString;
	response	: Tc2_System.T_MaxString;
END_VAR
VAR
	i	: int;
END_VAR
FOR i := 0 TO 99 BY 1 DO
	// Limit looping not to abuse PLC task
	IF _errorBuffer[i].ResponseErrorInfo = E_LaudaResponseError.NO_ERROR AND _errorBuffer[i].SendCommand = '' THEN
		EXIT;
	END_IF
	_errorBuffer[i] := _errorBuffer[i + 1];
END_FOR

_errorBuffer[0].SendCommand := sendCommand;
_errorBuffer[0].ResponseErrorInfo := LaudaHelper.ParseResponseError(Response := response);

_error := TRUE;
END_METHOD

METHOD PRIVATE DequeueCommand
VAR_INPUT
END_VAR

VAR
	i	: INT;
END_VAR
FOR i := 0 TO 99 BY 1 DO
	arrCommandBuffer[i] := arrCommandBuffer[i+1];
	IF i = 99 THEN
		arrCommandBuffer[100] := '';
	END_IF
END_FOR
END_METHOD

METHOD PRIVATE EnqueueCommand
VAR_INPUT
	Command	: Tc2_System.T_MaxString;
END_VAR

VAR
	i	: UINT;
	commandExistsButValueDiffer	: BOOL;
END_VAR
FOR i := 0 TO 100 BY 1 DO
	// If finding an empty or same command in queue, enter it here
	IF arrCommandBuffer[i] = '' OR arrCommandBuffer[i] = Command THEN
		arrCommandBuffer[i] := Command;
		EXIT;
	END_IF
END_FOR
END_METHOD

{attribute 'monitoring' := 'variable'}
// Collection of actual values reported back from Lauda device
PROPERTY PUBLIC ActualValues : REFERENCE TO ST_LaudaActualValuesCollection
GET
ActualValues ref= _actualValues;
END_GET
END_PROPERTY

{attribute 'monitoring' := 'variable'}
// Gets or sets various communication specific parameters
PROPERTY CommParameters : REFERENCE TO ST_LaudaCommParameters
GET
CommParameters ref= _commParameters;
END_GET
SET
_commParameters := CommParameters;
END_SET
END_PROPERTY

// Gets the fault diagnosis from Lauda
PROPERTY DeviceFaultDiagnosis : REFERENCE TO ST_LaudaFaults
GET
DeviceFaultDiagnosis ref= _faults;
END_GET
END_PROPERTY

{attribute 'monitoring' := 'variable'}
// Error flag, provided if there was an error with the Tcp connection 
// or the response from the device was not valid (error response).
PROPERTY Error : BOOL
GET
Error := _error;
END_GET
END_PROPERTY

// Gets the error buffer, containing last 100 send commands that were parsed returning an error.
PROPERTY ErrorBuffer : REFERENCE TO ARRAY[0..100] OF ST_LaudaReadWriteError
GET
ErrorBuffer := _errorBuffer;
END_GET
END_PROPERTY

// Gets the faults from the device. If fault status is TRUE, it means that particular fault is active.
PROPERTY Faults : REFERENCE TO ST_LaudaFaults
GET
Faults ref= _faults;
END_GET
END_PROPERTY

{attribute 'monitoring' := 'variable'}
// TcpIp connection status, TRUE if connected
PROPERTY PUBLIC TcpIpConnectionEstablished : BOOL
GET
TcpIpConnectionEstablished := _tcpIpConnectionEstablished;
END_GET
END_PROPERTY

END_FUNCTION_BLOCK

// TESTS/Test suites/FB_LaudaHelperTests
FUNCTION_BLOCK INTERNAL FB_LaudaHelperTests EXTENDS FB_TestSuite
VAR_INPUT
END_VAR
VAR_OUTPUT
END_VAR
VAR
	fbLauda	: FB_LaudaPro_P20(8);
	COMMAND_SUFFIX				: STRING := '$R$L';
	SEND_COMMAND_RESPONSE_OK	: STRING := 'OK';
	READ_COMMAND_RESPONSE_NOK	: STRING := 'ERR_'; 
END_VAR

Test01_AddSuffix();
Test02_RemoveSuffix();
Test03_ValidateReadCommandResponse();
Test04_ValidateSendCommandResponse();
Test05_ParseFault();
Test06_ParseResponseError();

METHOD Test01_AddSuffix
VAR_INPUT
END_VAR
VAR
	noSuffix			: STRING := 'suffixMissing';
	shouldHaveSuffix	: STRING;	
END_VAR
TcUnit.TEST('Test01_AddSuffix');

shouldHaveSuffix := LaudaHelper.AddSuffix(sData := noSuffix);

AssertEquals_STRING(
	Actual := shouldHaveSuffix,
	Expected := 'suffixMissing$R$L',
	Message := 'Adding suffix to the command should result in $R$L added to the end of the given string!');
	
TcUnit.TEST_FINISHED();
END_METHOD

METHOD Test02_RemoveSuffix
VAR_INPUT
END_VAR
VAR
	hasSuffix			: STRING := Tc2_Standard.CONCAT('iHaveSuffix', COMMAND_SUFFIX);
	shouldHaveNoSuffix	: STRING;	
END_VAR
TcUnit.TEST('Test02_RemoveSuffix');

shouldHaveNoSuffix := LaudaHelper.RemoveSuffix(sData := hasSuffix);

AssertEquals_STRING(
	Actual := shouldHaveNoSuffix,
	Expected := 'iHaveSuffix',
	Message := 'Removing suffix from the command should result in $R$L removed from the given string!');
	
TcUnit.TEST_FINISHED();
END_METHOD

METHOD Test03_ValidateReadCommandResponse
VAR_INPUT
END_VAR

VAR
	responseOk			: STRING := '55$R$L';
	responseNok			: STRING := '55_ERR_4$R$L';
	responseOkNoSuffix	: STRING := '55';
	responseNokNoSuffix	: STRING := '55_ERR_8';
END_VAR
TcUnit.TEST('Test03_ValidateReadCommandResponse');

AssertTrue(
	Condition := LaudaHelper.ValidateReadCommandResponse(responseOk),
	Message := 'Message without any ERR_ and with suffix $R$L is a valid read response!');

AssertFalse(
	Condition := LaudaHelper.ValidateReadCommandResponse(responseNok),
	Message :=  '55_ERR_4$R$L is considered invalid due to ERR_!');	
	
AssertFalse(
	Condition := LaudaHelper.ValidateReadCommandResponse(responseOkNoSuffix),
	Message :=  '55 is considered invalid due to no suffix ($R$L)!');	

AssertFalse(
	Condition := LaudaHelper.ValidateReadCommandResponse(responseNokNoSuffix),
	Message :=  '55_ERR_8 is considered invalid due to ERR_ and no suffix ($R$L)!');
		
TcUnit.TEST_FINISHED();
END_METHOD

METHOD Test04_ValidateSendCommandResponse
VAR_INPUT
END_VAR

VAR
	responseOk			: STRING := 'OK$R$L';
	responseOkNoSuffix	: STRING := 'OK';
	responseNok			: STRING := '__$R$L';
	responseNokNoSuffix	: STRING := '__';
END_VAR
TcUnit.TEST('Test04_ValidateSendCommandResponse');

AssertTrue(
	Condition := LaudaHelper.ValidateSendCommandResponse(responseOk),
	Message := 'OK$R$L should be a valid response!');
	
AssertFalse(
	Condition := LaudaHelper.ValidateSendCommandResponse(responseOkNoSuffix),
	Message := 'OK is invalid response due to missing suffix in the response string!');	

AssertFalse(
	Condition := LaudaHelper.ValidateSendCommandResponse(responseNok),
	Message := '__$R$L is invalid response due to missing OK in the response string!');
	
AssertFalse(
	Condition := LaudaHelper.ValidateSendCommandResponse(responseNokNoSuffix),
	Message := '__ is invalid response due to missing OK and missing suffix in the response string!');

TcUnit.TEST_FINISHED();
END_METHOD

METHOD Test05_ParseFault
VAR_INPUT
END_VAR
VAR
	laudaFaultsExpected	: ST_LaudaFaults;
	laudaFaultsActual	: ST_LaudaFaults;
END_VAR
TcUnit.TEST('Test05_ParseFault');
(* Fault is detected by looking at positions in the response string with the 7 digit value
XXXXXXX, if any of the valu is not 0, it inidicates the fault is active for that particular fault index
1 -> Error
2 -> Alarm
3 -> Warning
4 -> Overtemp
5 -> sublevel
6 -> higherLevel
7 -> ExternalControlValueMissing*)

laudaFaultsExpected.Error := FALSE;
laudaFaultsExpected.Alarm := FALSE;
laudaFaultsExpected.Warning := FALSE;
laudaFaultsExpected.Overtemp := FALSE;
laudaFaultsExpected.Sublevel := FALSE;
laudaFaultsExpected.HigherLevel := FALSE;
laudaFaultsExpected.ExternalControlValueMissing := FALSE;
laudaFaultsActual := LaudaHelper.ParseLaudaFaultDiagnosis(sDiagnosisResposne := '0000000$R$L');
AssertEquals(
	Expected := laudaFaultsExpected,
	Actual := laudaFaultsActual,
	Message := '0000000$R$L should have no faults active!');
	
laudaFaultsExpected.Error := TRUE;
laudaFaultsExpected.Alarm := FALSE;
laudaFaultsExpected.Warning := FALSE;
laudaFaultsExpected.Overtemp := FALSE;
laudaFaultsExpected.Sublevel := FALSE;
laudaFaultsExpected.HigherLevel := FALSE;
laudaFaultsExpected.ExternalControlValueMissing := FALSE;
laudaFaultsActual := LaudaHelper.ParseLaudaFaultDiagnosis(sDiagnosisResposne := '1000000$R$L');
AssertEquals(
	Expected := laudaFaultsExpected,
	Actual := laudaFaultsActual,
	Message := '1000000$R$L should have Error fault set to TRUE!');
	
laudaFaultsExpected.Error := FALSE;
laudaFaultsExpected.Alarm := TRUE;
laudaFaultsExpected.Warning := FALSE;
laudaFaultsExpected.Overtemp := FALSE;
laudaFaultsExpected.Sublevel := FALSE;
laudaFaultsExpected.HigherLevel := FALSE;
laudaFaultsExpected.ExternalControlValueMissing := FALSE;
laudaFaultsActual := LaudaHelper.ParseLaudaFaultDiagnosis(sDiagnosisResposne := '0100000$R$L');
AssertEquals(
	Expected := laudaFaultsExpected,
	Actual := laudaFaultsActual,
	Message := '0100000$R$L should have Alarm fault set to TRUE!');
	
laudaFaultsExpected.Error := FALSE;
laudaFaultsExpected.Alarm := FALSE;
laudaFaultsExpected.Warning := TRUE;
laudaFaultsExpected.Overtemp := FALSE;
laudaFaultsExpected.Sublevel := FALSE;
laudaFaultsExpected.HigherLevel := FALSE;
laudaFaultsExpected.ExternalControlValueMissing := FALSE;
laudaFaultsActual := LaudaHelper.ParseLaudaFaultDiagnosis(sDiagnosisResposne := '0010000$R$L');
AssertEquals(
	Expected := laudaFaultsExpected,
	Actual := laudaFaultsActual,
	Message := '00100000$R$L should have Warning fault set to TRUE!');

laudaFaultsExpected.Error := FALSE;
laudaFaultsExpected.Alarm := FALSE;
laudaFaultsExpected.Warning := FALSE;
laudaFaultsExpected.Overtemp := TRUE;
laudaFaultsExpected.Sublevel := FALSE;
laudaFaultsExpected.HigherLevel := FALSE;
laudaFaultsExpected.ExternalControlValueMissing := FALSE;
laudaFaultsActual := LaudaHelper.ParseLaudaFaultDiagnosis(sDiagnosisResposne := '0001000$R$L');
AssertEquals(
	Expected := laudaFaultsExpected,
	Actual := laudaFaultsActual,
	Message := '0001000$R$L should have Overtemp fault set to TRUE!');	
	
laudaFaultsExpected.Error := FALSE;
laudaFaultsExpected.Alarm := FALSE;
laudaFaultsExpected.Warning := FALSE;
laudaFaultsExpected.Overtemp := FALSE;
laudaFaultsExpected.Sublevel := TRUE;
laudaFaultsExpected.HigherLevel := FALSE;
laudaFaultsExpected.ExternalControlValueMissing := FALSE;
laudaFaultsActual := LaudaHelper.ParseLaudaFaultDiagnosis(sDiagnosisResposne := '0000100$R$L');
AssertEquals(
	Expected := laudaFaultsExpected,
	Actual := laudaFaultsActual,
	Message := '0000100$R$L should have Sublevel fault set to TRUE!');	

laudaFaultsExpected.Error := FALSE;
laudaFaultsExpected.Alarm := FALSE;
laudaFaultsExpected.Warning := FALSE;
laudaFaultsExpected.Overtemp := FALSE;
laudaFaultsExpected.Sublevel := FALSE;
laudaFaultsExpected.HigherLevel := TRUE;
laudaFaultsExpected.ExternalControlValueMissing := FALSE;
laudaFaultsActual := LaudaHelper.ParseLaudaFaultDiagnosis(sDiagnosisResposne := '0000010$R$L');
AssertEquals(
	Expected := laudaFaultsExpected,
	Actual := laudaFaultsActual,
	Message := '0000010$R$L should have HigherLevel fault set to TRUE!');	
	
laudaFaultsExpected.Error := FALSE;
laudaFaultsExpected.Alarm := FALSE;
laudaFaultsExpected.Warning := FALSE;
laudaFaultsExpected.Overtemp := FALSE;
laudaFaultsExpected.Sublevel := FALSE;
laudaFaultsExpected.HigherLevel := FALSE;
laudaFaultsExpected.ExternalControlValueMissing := TRUE;
laudaFaultsActual := LaudaHelper.ParseLaudaFaultDiagnosis(sDiagnosisResposne := '0000001$R$L');
AssertEquals(
	Expected := laudaFaultsExpected,
	Actual := laudaFaultsActual,
	Message := '0000001$R$L should have ExternalControlValueMissing fault set to TRUE!');

	
TcUnit.TEST_FINISHED();
END_METHOD

METHOD Test06_ParseResponseError
VAR_INPUT
END_VAR

VAR
	WrongEntry	 								: STRING := 'ERR_2';
	WrongCommand								: STRING := 'ERR_3';
	SyntaxError	 								: STRING := 'ERR_5';
	ImpermissableValue	 						: STRING := 'ERR_6';
	ModuleOrValueNotAvailable					: STRING := 'ERR_8';
	AllSegmentsInTheProgrammerAreOccupied		: STRING := 'ERR_30';
	SetpointNotPossible_AnalogSetpointIsUsed	: STRING := 'ERR_31';
	ExternalTemperatureProbeMissing	 			: STRING := 'ERR_33';
	AnalogValueNotPresent	 					: STRING := 'ERR_34';
	SafetyModeCantBeStarted_ItIsNotEnabled	 	: STRING := 'ERR_35';
	CantSetValue_ProgrammerRunningOrPaused	 	: STRING := 'ERR_36';
	CantStartProgrammer_AnalogSetpointIsUsed	: STRING := 'ERR_37';
	CantActivateFromSafetyMode	 				: STRING := 'ERR_38';
	
	parsedResponseActual	: E_LaudaResponseError;
	parsedResponseExpected	: E_LaudaResponseError;
END_VAR
TcUnit.TEST('Test06_ParseResponseError');

parsedResponseActual := LaudaHelper.ParseResponseError(WrongEntry);
parsedResponseExpected := E_LaudaResponseError.WRONG_ENTRY;
AssertEquals(
	Actual := parsedResponseActual,
	Expected := parsedResponseExpected,
	Message := Tc2_Standard.CONCAT('Invalid value returned for response with', WrongEntry));


parsedResponseActual := LaudaHelper.ParseResponseError(WrongCommand);
parsedResponseExpected := E_LaudaResponseError.WRONG_COMMAND;
AssertEquals(
	Actual := parsedResponseActual,
	Expected := parsedResponseExpected,
	Message := Tc2_Standard.CONCAT('Invalid value returned for response with', WrongCommand));


parsedResponseActual := LaudaHelper.ParseResponseError(SyntaxError);
parsedResponseExpected := E_LaudaResponseError.SYNTAX_ERROR;
AssertEquals(
	Actual := parsedResponseActual,
	Expected := parsedResponseExpected,
	Message := Tc2_Standard.CONCAT('Invalid value returned for response with', SyntaxError));


parsedResponseActual := LaudaHelper.ParseResponseError(ImpermissableValue);
parsedResponseExpected := E_LaudaResponseError.IMPERMISSABLE_VALUE;
AssertEquals(
	Actual := parsedResponseActual,
	Expected := parsedResponseExpected,
	Message := Tc2_Standard.CONCAT('Invalid value returned for response with', ImpermissableValue));


parsedResponseActual := LaudaHelper.ParseResponseError(ModuleOrValueNotAvailable);
parsedResponseExpected := E_LaudaResponseError.MODULE_OR_VALUE_NOT_AVAILABLE;
AssertEquals(
	Actual := parsedResponseActual,
	Expected := parsedResponseExpected,
	Message := Tc2_Standard.CONCAT('Invalid value returned for response with', ModuleOrValueNotAvailable));


parsedResponseActual := LaudaHelper.ParseResponseError(AllSegmentsInTheProgrammerAreOccupied);
parsedResponseExpected := E_LaudaResponseError.ALL_SEGMENTS_IN_THE_PROGRAMMER_OCCUPIED;
AssertEquals(
	Actual := parsedResponseActual,
	Expected := parsedResponseExpected,
	Message := Tc2_Standard.CONCAT('Invalid value returned for response with', AllSegmentsInTheProgrammerAreOccupied));


parsedResponseActual := LaudaHelper.ParseResponseError(SetpointNotPossible_AnalogSetpointIsUsed);
parsedResponseExpected := E_LaudaResponseError.SETPOINT_NOT_POSSIBLE_WITH_ANALOG_SETPOINT_USED;
AssertEquals(
	Actual := parsedResponseActual,
	Expected := parsedResponseExpected,
	Message := Tc2_Standard.CONCAT('Invalid value returned for response with', SetpointNotPossible_AnalogSetpointIsUsed));


parsedResponseActual := LaudaHelper.ParseResponseError(ExternalTemperatureProbeMissing);
parsedResponseExpected := E_LaudaResponseError.EXTERNAL_TEMPERATURE_PROBE_MISSING;
AssertEquals(
	Actual := parsedResponseActual,
	Expected := parsedResponseExpected,
	Message := Tc2_Standard.CONCAT('Invalid value returned for response with', ExternalTemperatureProbeMissing));


parsedResponseActual := LaudaHelper.ParseResponseError(AnalogValueNotPresent);
parsedResponseExpected := E_LaudaResponseError.ANALOG_VALUE_NOT_PRESENT;
AssertEquals(
	Actual := parsedResponseActual,
	Expected := parsedResponseExpected,
	Message := Tc2_Standard.CONCAT('Invalid value returned for response with', AnalogValueNotPresent));


parsedResponseActual := LaudaHelper.ParseResponseError(SafetyModeCantBeStarted_ItIsNotEnabled);
parsedResponseExpected := E_LaudaResponseError.SAFETY_MODE_CANT_START_IF_NOT_ENABLED;
AssertEquals(
	Actual := parsedResponseActual,
	Expected := parsedResponseExpected,
	Message := Tc2_Standard.CONCAT('Invalid value returned for response with', SafetyModeCantBeStarted_ItIsNotEnabled));


parsedResponseActual := LaudaHelper.ParseResponseError(CantSetValue_ProgrammerRunningOrPaused);
parsedResponseExpected := E_LaudaResponseError.CANT_SET_VALUE_PROGRAMMER_RUNNING_OR_PAUSED;
AssertEquals(
	Actual := parsedResponseActual,
	Expected := parsedResponseExpected,
	Message := Tc2_Standard.CONCAT('Invalid value returned for response with', CantSetValue_ProgrammerRunningOrPaused));


parsedResponseActual := LaudaHelper.ParseResponseError(CantStartProgrammer_AnalogSetpointIsUsed);
parsedResponseExpected := E_LaudaResponseError.CANT_START_PROGRAMMER_ANALOG_SETPOINT_USED;
AssertEquals(
	Actual := parsedResponseActual,
	Expected := parsedResponseExpected,
	Message := Tc2_Standard.CONCAT('Invalid value returned for response with', CantStartProgrammer_AnalogSetpointIsUsed));

parsedResponseActual := LaudaHelper.ParseResponseError(CantActivateFromSafetyMode);
parsedResponseExpected := E_LaudaResponseError.CANT_ACTIVATE_FROM_SAFETY_MODE;
AssertEquals(
	Actual := parsedResponseActual,
	Expected := parsedResponseExpected,
	Message := Tc2_Standard.CONCAT('Invalid value returned for response with', CantActivateFromSafetyMode));
TcUnit.TEST_FINISHED();
END_METHOD

END_FUNCTION_BLOCK

// TESTS/PRG_TESTS
PROGRAM INTERNAL PRG_TESTS

(* Instantiate test suites here. Naming convention for tests should be a suffix with _Tests.
Good practice for creating test methods is to end them with _test as well. *)
VAR
	LaudaHelperTest	: FB_LaudaHelperTests;

END_VAR

// Run tests in paralel
TcUnit.RUN();

// Run tests in sequence, one after the other. Uncomment if required.
// TcUnit.RUN_IN_SEQUENCE();

END_PROGRAM
